FUNCTION_BLOCK FG_02

{region generated code}
VAR_INPUT
	P_Camera : FB_Camera;
END_VAR
{endregion}

{region generated code}
	InitRun();
	P_Camera();
{endregion}

METHOD InitRun
{region generated code}
VAR_INST
	bInitRun : BOOL := TRUE;
END_VAR
{endregion}
{region generated code}
	IF NOT bInitRun THEN RETURN; END_IF
	bInitRun := FALSE;
{endregion}
END_METHOD

END_FUNCTION_BLOCK

(* stored: Version 1.1.0.1, ProductVersion 3.1.4026.19
   POU FG_02: Id {669b5fb7-101c-4b47-8f64-4b0c099808fe}, SpecialFunc None
   Method InitRun: Id {9f43e803-fcdb-4fb1-81ce-65421d04daeb} *)
